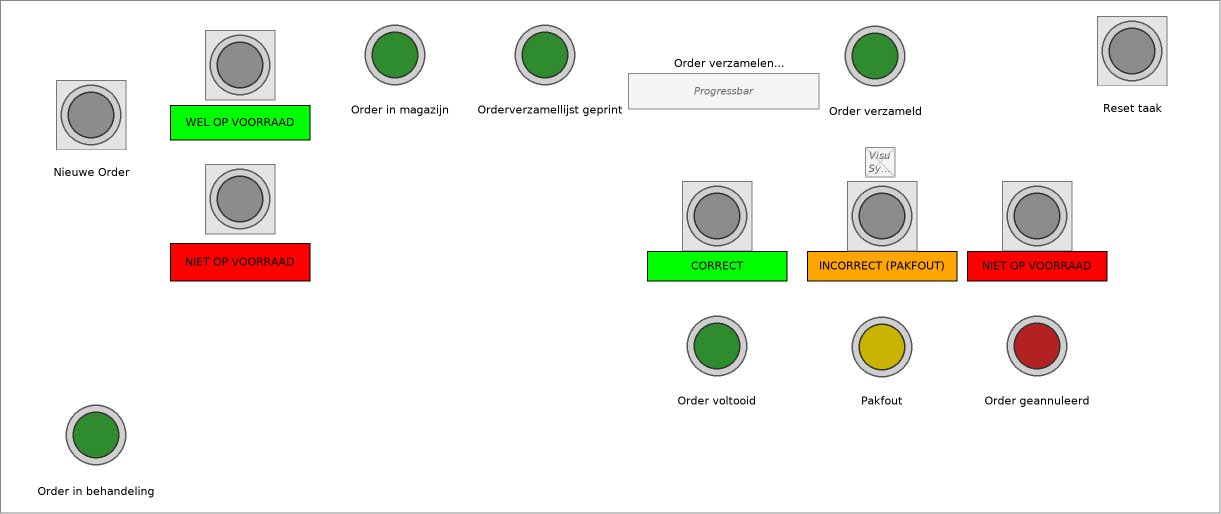
VISUALIZATION Orderverwerking_magazijn  // 1221x514
    Group (170,30 140x250)
        PushSwitch (35,0 70x70), variable: Orderverwerking_magazijn.WelOpVoorraad, behaviour: TOGGLE, style: Switch-PushSwitch-Gray
        Rectangle (0,75 140x35), "WEL OP VOORRAAD"
        PushSwitch (35,134 70x70), variable: Orderverwerking_magazijn.NietOpVoorraad, behaviour: TOGGLE, style: Switch-PushSwitch-Gray
        Rectangle (0,213 140x38), "NIET OP VOORRAAD"
    Group (30,80 120x110)
        PushSwitch (26,0 70x70), variable: Orderverwerking_magazijn.Nieuwe_order, behaviour: TOGGLE, style: Switch-PushSwitch-Gray
        Rectangle (0,70 123x45), "Nieuwe Order"
    Lamp1 (360,20 70x70), variable: Orderverwerking_magazijn.Order_magazijn, style: Lamp-Lamp1-Green
    Rectangle (340,90 120x40), "Order in magazijn"
    Lamp1 (510,20 70x70), variable: Orderverwerking_magazijn.Order_uitgeprint, style: Lamp-Lamp1-Green
    Rectangle (460,90 180x40), "Orderverzamellijst geprint"
    Group (21,400 150x114)
        Lamp1 (40,0 70x70), variable: Orderverwerking_magazijn.Nieuwe_order, style: Lamp-Lamp1-Green
        Rectangle (0,69 150x45), "Order in behandeling"
    Group (787,21 180x110)
        Lamp1 (53,0 70x70), variable: Orderverwerking_magazijn.Order_verzameld, style: Lamp-Lamp1-Green
        Rectangle (0,68 177x45), "Order verzameld"
    Group (628,41 190x70)
        Rectangle (13,0 177x45), "Order verzamelen..."
        Progressbar (0,32 191x36), variable: Orderverwerking_magazijn.WachtTijd
    Group (627,181 480x240)
        Group (335,130 150x110)
            Lamp1 (40,0 70x70), variable: Orderverwerking_magazijn.Geannuleerd, style: Lamp-Lamp1-Red
            Rectangle (0,70 150x40), "Order geannuleerd"
        Group (20,0 140x100)
            PushSwitch (35,0 70x70), variable: Orderverwerking_magazijn.Correct, behaviour: TAP, style: Switch-PushSwitch-Gray
            Rectangle (0,70 140x30), "CORRECT"
        Group (180,0 150x100)
            Rectangle (0,70 150x30), "INCORRECT (PAKFOUT)"
            PushSwitch (40,0 70x70), variable: Orderverwerking_magazijn.Pakfout, behaviour: TOGGLE, style: Switch-PushSwitch-Gray
        Group (340,0 140x100)
            PushSwitch (35,0 70x70), variable: Orderverwerking_magazijn.Incorrect, behaviour: TAP, style: Switch-PushSwitch-Gray
            Rectangle (0,70 140x30), "NIET OP VOORRAAD"
        Group (0,130 180x110)
            Lamp1 (55,0 70x70), variable: Orderverwerking_magazijn.Order_voltooid, style: Lamp-Lamp1-Green
            Rectangle (0,70 180x40), "Order voltooid"
        Group (165,131 180x109)
            Lamp1 (55,0 70x70), variable: Orderverwerking_magazijn.Pakfout, style: Lamp-Lamp1-Yellow
            Rectangle (0,69 180x40), "Pakfout"
    Group (1044,16 177x115)
        PushSwitch (53,0 70x70), variable: Orderverwerking_magazijn.Taak1Reset, behaviour: TAP, style: Switch-PushSwitch-Gray
        Rectangle (0,70 177x45), "Reset taak"
    Image (865,147 30x30), image: VisuSymbols.Symbols.ArrowBoldDown
END_VISUALIZATION

(* stored: Version 1.1.0.1, ProductVersion 3.1.4024.12
   Visu Orderverwerking_magazijn: Id {34a5ba20-7505-44f5-9032-92cf551bd65b} *)
